// TIA Portal V19 export
FUNCTION "M_PosAPlusCostB" : LReal   // FC34, LAD
TITLE = Module POSA plus CostantB / Position A plus Costant B
// stored: Access Published, SetENOAutomatically false
   VAR_INPUT
      PosA : LReal;
      CostB : LReal;
      MODULE : LReal;
   END_VAR
   VAR_TEMP
      Xc : LReal;
   END_VAR
BEGIN

REGION Network 1 (SCL): Xc = PosA + CostB / Main
   #Xc := #PosA + #CostB;
   #M_PosAPlusCostB := #Xc;

   IF #MODULE > 0.0 THEN

       IF #Xc >= #MODULE THEN
           #M_PosAPlusCostB := #Xc - #MODULE;
       ELSIF #Xc < 0 THEN
           #M_PosAPlusCostB := #MODULE + #Xc;
       END_IF;

       IF ABS(#M_PosAPlusCostB - #MODULE) < 0.01 THEN
           #M_PosAPlusCostB := 0;
       END_IF;

   END_IF;
END_REGION
END_FUNCTION
